% RSLogix 500 project pump prog.RSS, saved by version 8.30.00.16 %
PROJECT "UNTITLED"    % processor: Bul.1763 MicroLogix 1100 Series B %

PROGRAM FILES
  LAD 2 "MAIN"  2 rungs
  LAD 3 "I/O"  10 rungs

DATA FILES
  O0 OUTPUT  5 elements
  I1 INPUT  7 elements
  S2 STATUS  66 elements
  B3 BINARY  1 elements
  T4 TIMER  3 elements
  C5 COUNTER  1 elements
  R6 CONTROL  1 elements
  N7 INTEGER  1 elements
  F8 FLOAT  1 elements

LADDER 2 "MAIN"
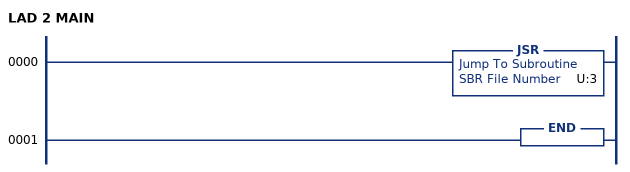
% Rung: 0 %
SOR JSR U:3 EOR
% Rung: 1 %
SOR END EOR

LADDER 3 "I/O"
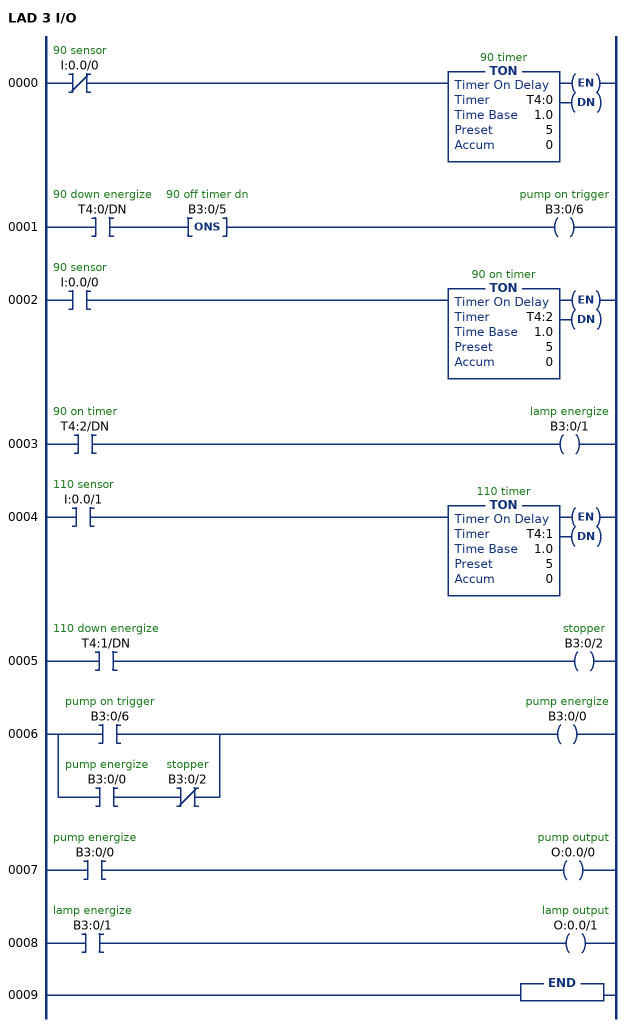
% Rung: 0 %
SOR XIO I:0.0/0 TON T4:0 1.0 5 0 EOR
%   I:0.0/0  "90 sensor" %
%   T4:0  "90 timer" %
% Rung: 1 %
SOR XIC T4:0/DN ONS B3:0/5 OTE B3:0/6 EOR
%   T4:0/DN  "90 down energize" %
%   B3:0/5  "90 off timer dn" %
%   B3:0/6  "pump on trigger" %
% Rung: 2 %
SOR XIC I:0.0/0 TON T4:2 1.0 5 0 EOR
%   I:0.0/0  "90 sensor" %
%   T4:2  "90 on timer" %
% Rung: 3 %
SOR XIC T4:2/DN OTE B3:0/1 EOR
%   T4:2/DN  "90 on timer" %
%   B3:0/1  "lamp energize" %
% Rung: 4 %
SOR XIC I:0.0/1 TON T4:1 1.0 5 0 EOR
%   I:0.0/1  "110 sensor" %
%   T4:1  "110 timer" %
% Rung: 5 %
SOR XIC T4:1/DN OTE B3:0/2 EOR
%   T4:1/DN  "110 down energize" %
%   B3:0/2  "stopper" %
% Rung: 6 %
SOR BST XIC B3:0/6 NXB XIC B3:0/0 XIO B3:0/2 BND OTE B3:0/0 EOR
%   B3:0/6  "pump on trigger" %
%   B3:0/0  "pump energize" %
%   B3:0/2  "stopper" %
% Rung: 7 %
SOR XIC B3:0/0 OTE O:0.0/0 EOR
%   B3:0/0  "pump energize" %
%   O:0.0/0  "pump output" %
% Rung: 8 %
SOR XIC B3:0/1 OTE O:0.0/1 EOR
%   B3:0/1  "lamp energize" %
%   O:0.0/1  "lamp output" %
% Rung: 9 %
SOR END EOR

OTHER DOCUMENTED ADDRESSES
  B3:0/4  "ons 90 on timer dn"
  B3:0/7  "110 on timer ons"
  T4:0/0  "90 timer"

DATA TABLE (non-zero values as saved)
DATA T4
% .PRE .ACC %
% T4:0 % 5 0
% T4:1 % 5 0
% T4:2 % 5 0
